PROGRAM NOVRAM
VAR
END_VAR

;

END_PROGRAM

(* stored: Version 1.1.0.1, ProductVersion 3.1.4024.10
   POU NOVRAM: Id {5d91f566-ba50-433e-8d55-1c9ba1ba3ec9}, SpecialFunc None *)
